(* PLC project PLC, Beckhoff Automation GmbH TwinCAT PLC Control 3.5.13.21 *)
(* stored: creationDateTime 2024-02-17T22:43:41.2426721, modificationDateTime 2024-02-17T22:43:41.2426721 *)

FUNCTION_BLOCK PB
VAR_INPUT
	index: LINT;
	name: STRING(G.nameStringLength);
END_VAR
VAR_OUTPUT
	pushed: BOOL;
END_VAR
VAR_IN_OUT
	resources: ARRAY[0..G.numAxis] OF PBResource;
END_VAR
VAR
	input: PBInput;
	config: PBConfig;
	status: PBStatus;
	TON_0: TON;
END_VAR

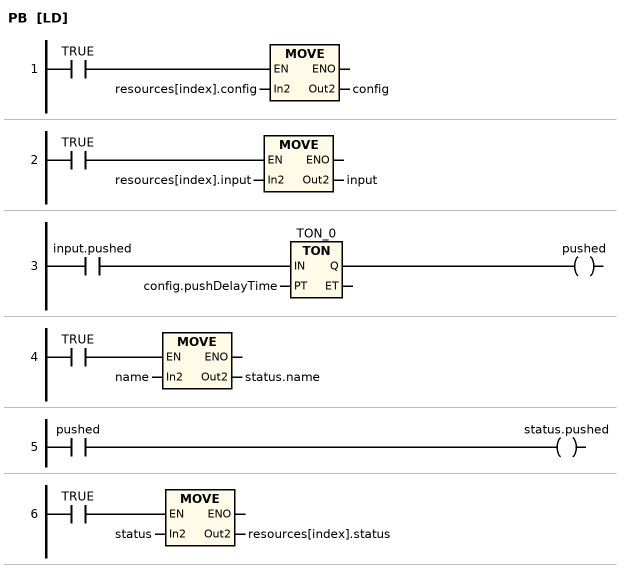
(* LD diagram, written out as Structured Text *)

IF TRUE THEN config := resources[index].config; END_IF;

IF TRUE THEN input := resources[index].input; END_IF;


TON_0(IN := input.pushed, PT := config.pushDelayTime);
pushed := TON_0.Q;

IF TRUE THEN status.name := name; END_IF;

status.pushed := pushed;

IF TRUE THEN resources[index].status := status; END_IF;
END_FUNCTION_BLOCK
